{attribute 'GeneratedUsingTerminal: EP7402-0057-0017'}
{attribute addProperty BoxType "EP7402-0057-0017"}
{attribute addProperty Id "Device_undervoltageBOOL1Device_overvoltageBOOL1Overtemperature_warningBOOL1Overtemperature_errorBOOL1General_hardware_errorBOOL1Channel_1_openloadBOOL1Channel_1_short_circuitBOOL1Channel_1_motor_overload_I2T_warningBOOL1Channel_1_motor_overload_I2T_errorBOOL1Channel_1_amplifier_overload_I2T_warningBOOL1Channel_1_amplifier_overload_I2T_errorBOOL1Channel_1_in_limit_xBOOL1Channel_1_commutation_errorBOOL1Channel_2_openloadBOOL1Channel_2_short_circuitBOOL1Channel_2_motor_overload_I2T_warningBOOL1Channel_2_motor_overload_I2T_errorBOOL1Channel_2_amplifier_overload_I2T_warningBOOL1Channel_2_amplifier_overload_I2T_errorBOOL1Channel_2_in_limit_xBOOL1Channel_2_commutation_errorBOOL1"}
{attribute addProperty CRC "342158585"}
{attribute addProperty Size "21"}
TYPE Device_Diag_1464ECF9 :
STRUCT
	{attribute addProperty Name "Device_undervoltage"}
	Device_undervoltage : BOOL;
	{attribute addProperty Name "Device_overvoltage"}
	Device_overvoltage : BOOL;
	{attribute addProperty Name "Overtemperature_warning"}
	Overtemperature_warning : BOOL;
	{attribute addProperty Name "Overtemperature_error"}
	Overtemperature_error : BOOL;
	{attribute addProperty Name "General_hardware_error"}
	General_hardware_error : BOOL;
	{attribute addProperty Name "Channel_1_openload"}
	Channel_1_openload : BOOL;
	{attribute addProperty Name "Channel_1_short_circuit"}
	Channel_1_short_circuit : BOOL;
	{attribute addProperty Name "Channel_1_motor_overload_I2T_warning"}
	Channel_1_motor_overload_I2T_warning : BOOL;
	{attribute addProperty Name "Channel_1_motor_overload_I2T_error"}
	Channel_1_motor_overload_I2T_error : BOOL;
	{attribute addProperty Name "Channel_1_amplifier_overload_I2T_warning"}
	Channel_1_amplifier_overload_I2T_warning : BOOL;
	{attribute addProperty Name "Channel_1_amplifier_overload_I2T_error"}
	Channel_1_amplifier_overload_I2T_error : BOOL;
	{attribute addProperty Name "Channel_1_in_limit_x"}
	Channel_1_in_limit_x : BOOL;
	{attribute addProperty Name "Channel_1_commutation_error"}
	Channel_1_commutation_error : BOOL;
	{attribute addProperty Name "Channel_2_openload"}
	Channel_2_openload : BOOL;
	{attribute addProperty Name "Channel_2_short_circuit"}
	Channel_2_short_circuit : BOOL;
	{attribute addProperty Name "Channel_2_motor_overload_I2T_warning"}
	Channel_2_motor_overload_I2T_warning : BOOL;
	{attribute addProperty Name "Channel_2_motor_overload_I2T_error"}
	Channel_2_motor_overload_I2T_error : BOOL;
	{attribute addProperty Name "Channel_2_amplifier_overload_I2T_warning"}
	Channel_2_amplifier_overload_I2T_warning : BOOL;
	{attribute addProperty Name "Channel_2_amplifier_overload_I2T_error"}
	Channel_2_amplifier_overload_I2T_error : BOOL;
	{attribute addProperty Name "Channel_2_in_limit_x"}
	Channel_2_in_limit_x : BOOL;
	{attribute addProperty Name "Channel_2_commutation_error"}
	Channel_2_commutation_error : BOOL;
END_STRUCT
END_TYPE

(* stored: Version 1.2.0.0, ProductVersion 3.1.4024.9
   DUT Device_Diag_1464ECF9: Id {dcc8f3f5-97aa-4d43-807a-123500b260cb} *)
